Staubli VAL3: remGetIP.pgx

program remGetIP(string& sReturn[] (dimensions=1))
begin
  // Return which interaction point is active.
  //
  logMsg("call remGetIP")
  sReturn="GETIP "+toString("",nIPNumber)
end
